{attribute 'reflection'}
FUNCTION_BLOCK FB_Station IMPLEMENTS IStation, IObject
VAR_INPUT
END_VAR
VAR_OUTPUT
END_VAR
VAR
    _Position          : REFERENCE TO FB_Position;
    _Process           : REFERENCE TO FB_AUT_ABSTRACT;
    _WaitPosOffset     : LREAL; // offset of the station position, should always be negative
    _iMaxWaitingMovers : INT;   // Maximum of waiting mover in front of the station
    _iGroupNumber      : INT;   // The current group member
    _lrOffset          : LREAL; // offset position of this station for a given recipe
    _bSuperTrackNumber : BYTE;  // target number in superTrack

    _ApproachScenario : ApproachScenario_e := ApproachScenario_e.WaitOnFinishedProcess;

    _iID : INT := 0; // instance ID, is set during FB_Init using the value of _iInstanceCounter 
END_VAR
VAR_STAT
    _iInstanceCounter : INT := 1; // instance counter
END_VAR

PROPERTY ApproachScenario : ApproachScenario_e
GET
ApproachScenario := THIS^._ApproachScenario;
END_GET
SET
THIS^._ApproachScenario := ApproachScenario;
END_SET
END_PROPERTY

METHOD Equals : BOOL
VAR_INPUT
    object : ANY;
END_VAR
Equals := THIS = object.pValue;
END_METHOD

METHOD FB_init : BOOL
VAR_INPUT
    bInitRetains      : BOOL; // if TRUE, the retain variables are initialized (warm start / cold start)
    bInCopyCode       : BOOL; // if TRUE, the instance afterwards gets moved into the copy code (online change)
    Position          : REFERENCE TO FB_Position;
    Process           : REFERENCE TO FB_AUT_ABSTRACT;
    WaitPosOffset     : LREAL;
    ApproachScenario  : ApproachScenario_e;
    iMaxWaitingMovers : INT;
	bSuperTrackNumber : BYTE;
END_VAR
THIS^._iID               := THIS^._iInstanceCounter;
THIS^._iInstanceCounter  := THIS^._iInstanceCounter + 1;
THIS^._Position          REF= Position;
THIS^._Process           REF= Process;
THIS^._WaitPosOffset     := WaitPosOffset;
THIS^._ApproachScenario  := ApproachScenario;
THIS^._iMaxWaitingMovers := iMaxWaitingMovers;
THIS^._bSuperTrackNumber := bSuperTrackNumber;
END_METHOD

// the maxuimum number of waiting movers at the front of the station
PROPERTY iMaxWaitingMovers : INT
GET
iMaxWaitingMovers := THIS^._iMaxWaitingMovers;
END_GET
SET
THIS^._iMaxWaitingMovers := iMaxWaitingMovers;
END_SET
END_PROPERTY

PROPERTY PUBLIC Offset : LREAL
GET
Offset := THIS^._lrOffset;
END_GET
SET
THIS^._lrOffset := Offset;
END_SET
END_PROPERTY

PROPERTY Position : REFERENCE TO FB_Position
GET
Position REF=_Position;
END_GET
SET
_Position REF=Position;
END_SET
END_PROPERTY

PROPERTY Process : REFERENCE TO FB_AUT_ABSTRACT
GET
Process REF=_Process;
END_GET
SET
_Process REF= Process;
END_SET
END_PROPERTY

METHOD SetWaitPosOffset : REFERENCE TO FB_Station
VAR_INPUT
	WaitPosOffset : LREAL; // offset position from the given station, must be negative
END_VAR
IF _WaitPosOffset < 0 THEN
    _WaitPosOffset := WaitPos;
END_IF

SetWaitPosOffset REF= THIS^;
END_METHOD

PROPERTY SuperTrackNumber : BYTE
GET
SuperTrackNumber := THIS^._bSuperTrackNumber;
END_GET
END_PROPERTY

METHOD ToString : STRING
VAR_INPUT
END_VAR
VAR_INST
END_VAR
ToString := CONCAT('FB_Station_', TO_STRING(THIS^._iID));
END_METHOD

PROPERTY PUBLIC WaitPos : LREAL
GET
WaitPos := _WaitPosOffset + this^._Position.lrWorkPosition;
END_GET
SET
IF WaitPos < THIS^._Position.lrWorkPosition THEN
    _WaitPosOffset := WaitPos - THIS^._Position.lrWorkPosition;
END_IF
END_SET
END_PROPERTY

END_FUNCTION_BLOCK

(* stored: Version 1.1.0.1, ProductVersion 3.1.4024.12
   POU FB_Station: Id {70468013-f9f1-48d7-8a41-9e3de9ebad9e}, SpecialFunc None
   Property ApproachScenario: Id {7af8662f-299f-4992-b910-3a98e1ea7f68}
   Get Get: Id {1e543aa0-4bf9-42e8-940f-25810da7807f}
   Set Set: Id {e2d8175a-d65d-404d-9515-d955dd39fe95}
   Method Equals: Id {8533c6eb-957c-422e-872a-afb3d6aaedc0}
   Method FB_init: Id {79a4bdc5-c74e-4221-9bda-a7d762e9f476}
   Property iMaxWaitingMovers: Id {546a0cb8-d5d0-4609-a889-24ff44d0a25e}
   Get Get: Id {4718007c-6aa3-4b8c-8d42-153f81de44ba}
   Set Set: Id {3ce85e75-a23d-47db-9068-e9fc275ba4d2}
   Property Offset: Id {0f5c0952-f6ae-4ee6-a98e-3ef72644cd22}
   Get Get: Id {a2b591ed-26cc-4237-a108-b54e2e588ae0}
   Set Set: Id {e6b836b5-2768-4f08-a3fe-d5e742cff61f}
   Property Position: Id {b6ed5e54-2fb9-44f3-99fb-44d690ace79e}
   Get Get: Id {d57d7b2c-d047-4546-b08e-9f2b19da1c3b}
   Set Set: Id {8ec541f4-51cc-47f8-8d1c-bda0126f4084}
   Property Process: Id {593b9bcf-49e5-4201-a417-8a170114a5c6}
   Get Get: Id {9be8e146-1278-4d03-b2c3-cc913e6cc63d}
   Set Set: Id {0b3f8467-e46f-497e-b2d6-a49d47d1d3ba}
   Method SetWaitPosOffset: Id {e4c044ad-097c-49d2-be32-46dd34cbd590}
   Property SuperTrackNumber: Id {48708baa-3e61-4dbb-9ae9-95a95949b98d}
   Get Get: Id {708941da-5b74-4ce8-aea6-ab99c1baa276}
   Method ToString: Id {efefe0e5-d9df-4b18-a791-065ec8f343b5}
   Property WaitPos: Id {8969891e-6d5a-4788-abdc-d61b00c916a8}
   Get Get: Id {4b1069d2-41b4-4948-8a2f-7c112e876a7c}
   Set Set: Id {0501bd4d-6f15-4e80-9d24-a4a4472e0372} *)
